FUNCTION_BLOCK EL6001
VAR
	_io : EL6001_Data;
	{attribute addProperty Name "WcState"}
	_wcState : WcStateInputToggle;
	{attribute addProperty Name "Info data"}
	_infoData : InfoDataAds;
END_VAR

PROPERTY IO : REFERENCE TO EL6001_Data
GET
IO REF= _io;
END_GET
END_PROPERTY

PROPERTY WcState : REFERENCE TO WcStateInputToggle
GET
WcState REF= _wcState;
END_GET
END_PROPERTY

END_FUNCTION_BLOCK

(* stored: Version 1.1.0.1, ProductVersion 3.1.4024.9
   POU EL6001: Id {d48c3dde-dfb9-0aeb-03c1-fbc82450b229}, SpecialFunc None
   Property IO: Id {fc582108-e0cb-03af-10cf-5cd379942ae3}
   Get Get: Id {5f480836-afc2-0608-2c83-9b5fae7d1af2}
   Property WcState: Id {f06591f6-fc9b-0d5c-294b-9f896083a16a}
   Get Get: Id {9a044e55-5ff5-00c6-2bb1-2dde0f934142} *)
